% RSLogix 500 project Sesion12_Tarea1_Josue Santana Robledo Corona.RSS, saved by version 8.40.00.08 %
PROJECT "UNTITLED"    % processor: MicroLogix 1200 %

PROGRAM FILES
  LAD 2 "MAIN"  7 rungs
  LAD 3 "ENTRADAS"  6 rungs
  LAD 4 "SALIDAS"  6 rungs
  LAD 5 "AUTOMATICO"  17 rungs
  LAD 6 "MANUAL"  6 rungs
  LAD 7 "HMI"  1 rungs
  LAD 8 "ALARMAS"  1 rungs
  LAD 9 "PARPADEOS"  9 rungs
  LAD 10 "RESETS"  7 rungs
  LAD 11 "LS"  3 rungs

DATA FILES
  O0 OUTPUT  4 elements
  I1 INPUT  4 elements
  S2 STATUS  66 elements
  B3 BINARY  5 elements
  T4 TIMER  7 elements
  C5 COUNTER  3 elements
  R6 CONTROL  1 elements
  N7 INTEGER  1 elements
  F8 FLOAT  1 elements

LADDER 2 "MAIN"
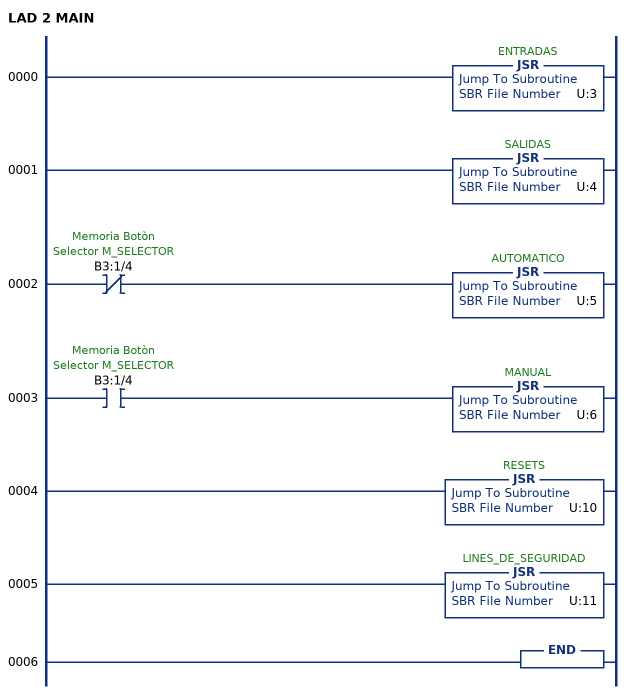
% Rung: 0 %
SOR JSR U:3 EOR
%   U:3  ENTRADAS %
% Rung: 1 %
SOR JSR U:4 EOR
%   U:4  SALIDAS %
% Rung: 2 %
SOR XIO B3:1/4 JSR U:5 EOR
%   B3:1/4  M_SELECTOR  "Memoria Botòn Selector" %
%   U:5  AUTOMATICO %
% Rung: 3 %
SOR XIC B3:1/4 JSR U:6 EOR
%   B3:1/4  M_SELECTOR  "Memoria Botòn Selector" %
%   U:6  MANUAL %
% Rung: 4 %
SOR JSR U:10 EOR
%   U:10  RESETS %
% Rung: 5 %
SOR JSR U:11 EOR
%   U:11  LINES_DE_SEGURIDAD %
% Rung: 6 %
SOR END EOR

LADDER 3 "ENTRADAS"
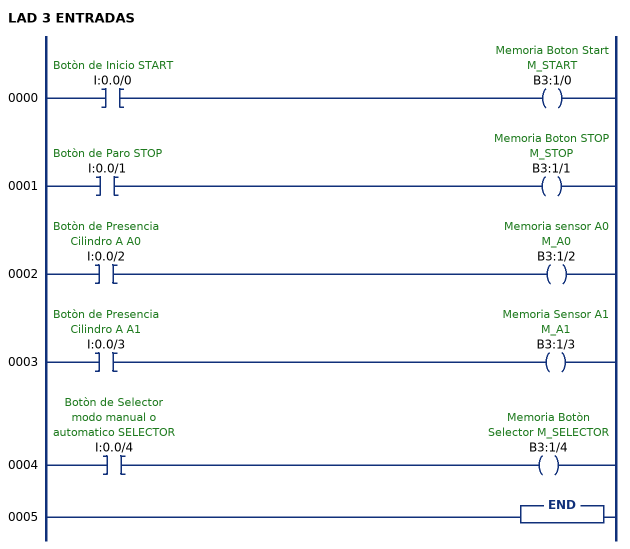
% Rung: 0 %
SOR XIC I:0.0/0 OTE B3:1/0 EOR
%   I:0.0/0  START  "Botòn de Inicio" %
%   B3:1/0  M_START  "Memoria Boton Start" %
% Rung: 1 %
SOR XIC I:0.0/1 OTE B3:1/1 EOR
%   I:0.0/1  STOP  "Botòn de Paro" %
%   B3:1/1  M_STOP  "Memoria Boton STOP" %
% Rung: 2 %
SOR XIC I:0.0/2 OTE B3:1/2 EOR
%   I:0.0/2  A0  "Botòn de Presencia Cilindro A" %
%   B3:1/2  M_A0  "Memoria sensor A0" %
% Rung: 3 %
SOR XIC I:0.0/3 OTE B3:1/3 EOR
%   I:0.0/3  A1  "Botòn de Presencia Cilindro A" %
%   B3:1/3  M_A1  "Memoria Sensor A1" %
% Rung: 4 %
SOR XIC I:0.0/4 OTE B3:1/4 EOR
%   I:0.0/4  SELECTOR  "Botòn de Selector modo manual o automatico" %
%   B3:1/4  M_SELECTOR  "Memoria Botòn Selector" %
% Rung: 5 %
SOR END EOR

LADDER 4 "SALIDAS"
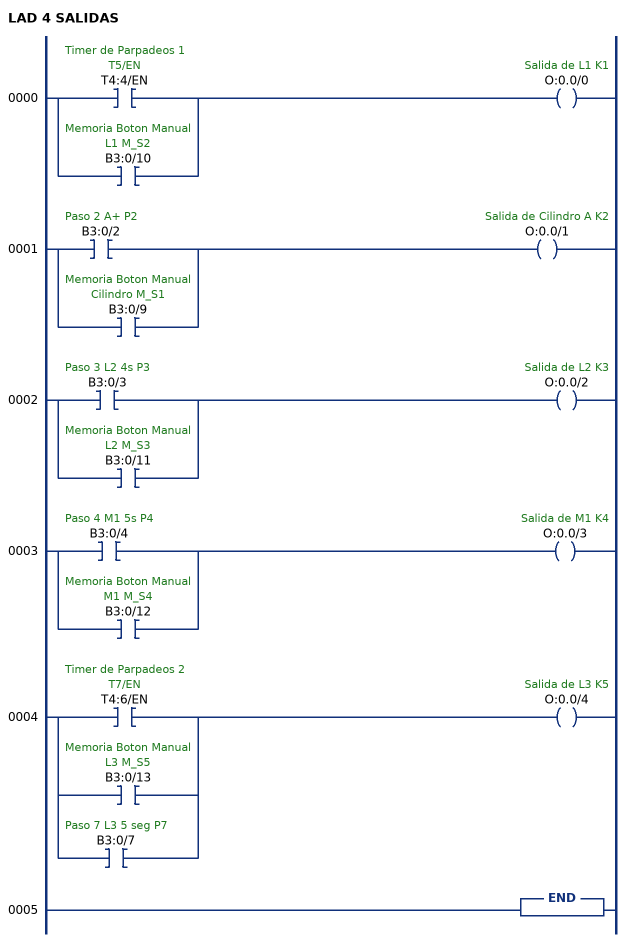
% Rung: 0 %
SOR BST XIC T4:4/EN NXB XIC B3:0/10 BND OTE O:0.0/0 EOR
%   T4:4  T5  "Timer de Parpadeos 1" %
%   B3:0/10  M_S2  "Memoria Boton Manual L1" %
%   O:0.0/0  K1  "Salida de L1" %
% Rung: 1 %
SOR BST XIC B3:0/2 NXB XIC B3:0/9 BND OTE O:0.0/1 EOR
%   B3:0/2  P2  "Paso 2 A+" %
%   B3:0/9  M_S1  "Memoria Boton Manual Cilindro" %
%   O:0.0/1  K2  "Salida de Cilindro A" %
% Rung: 2 %
SOR BST XIC B3:0/3 NXB XIC B3:0/11 BND OTE O:0.0/2 EOR
%   B3:0/3  P3  "Paso 3 L2 4s" %
%   B3:0/11  M_S3  "Memoria Boton Manual L2" %
%   O:0.0/2  K3  "Salida de L2" %
% Rung: 3 %
SOR BST XIC B3:0/4 NXB XIC B3:0/12 BND OTE O:0.0/3 EOR
%   B3:0/4  P4  "Paso 4 M1 5s" %
%   B3:0/12  M_S4  "Memoria Boton Manual M1" %
%   O:0.0/3  K4  "Salida de M1" %
% Rung: 4 %
SOR BST XIC T4:6/EN NXB XIC B3:0/13 NXB XIC B3:0/7 BND OTE O:0.0/4 EOR
%   T4:6  T7  "Timer de Parpadeos 2" %
%   B3:0/13  M_S5  "Memoria Boton Manual L3" %
%   B3:0/7  P7  "Paso 7 L3 5 seg" %
%   O:0.0/4  K5  "Salida de L3" %
% Rung: 5 %
SOR END EOR

LADDER 5 "AUTOMATICO"
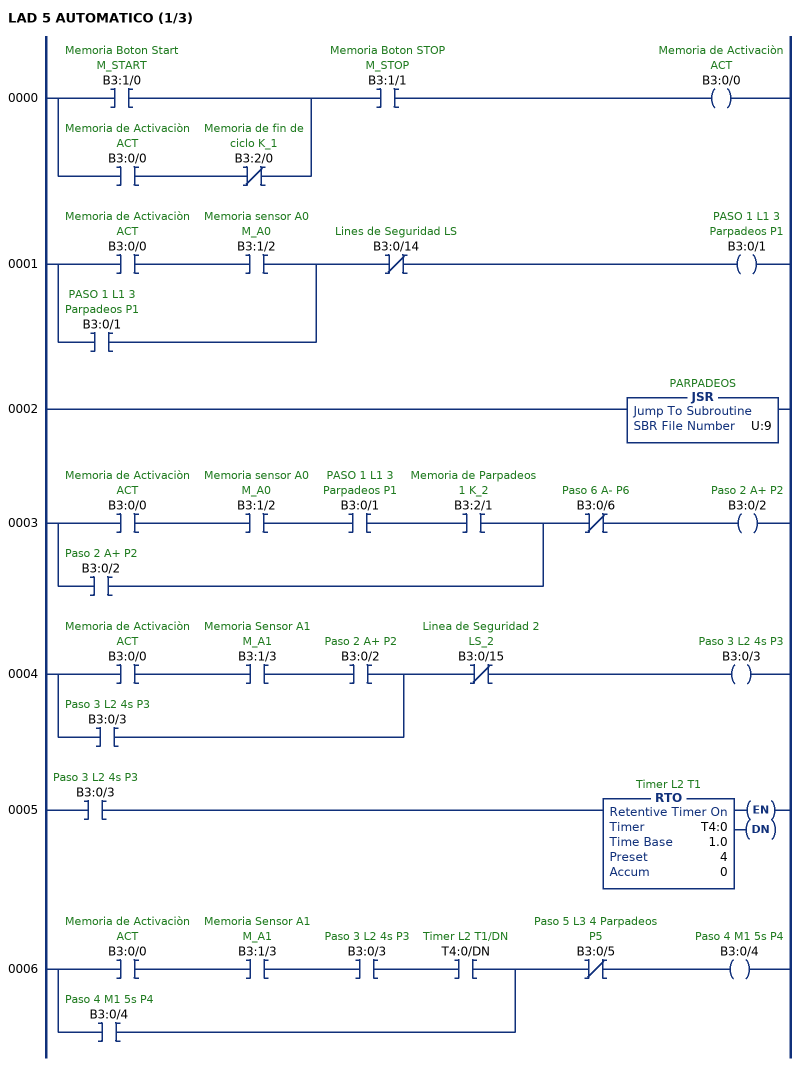
% Rung: 0 %
SOR BST XIC B3:1/0 NXB XIC B3:0/0 XIO B3:2/0 BND XIC B3:1/1 OTE B3:0/0 EOR
%   B3:1/0  M_START  "Memoria Boton Start" %
%   B3:0/0  ACT  "Memoria de Activaciòn" %
%   B3:2/0  K_1  "Memoria de fin de ciclo" %
%   B3:1/1  M_STOP  "Memoria Boton STOP" %
% Rung: 1 %
SOR BST XIC B3:0/0 XIC B3:1/2 NXB XIC B3:0/1 BND XIO B3:0/14 OTE B3:0/1 EOR
%   B3:0/0  ACT  "Memoria de Activaciòn" %
%   B3:1/2  M_A0  "Memoria sensor A0" %
%   B3:0/1  P1  "PASO 1 L1 3 Parpadeos" %
%   B3:0/14  LS  "Lines de Seguridad" %
% Rung: 2 %
SOR JSR U:9 EOR
%   U:9  PARPADEOS %
% Rung: 3 %
SOR BST XIC B3:0/0 XIC B3:1/2 XIC B3:0/1 XIC B3:2/1 NXB XIC B3:0/2 BND XIO B3:0/6 OTE B3:0/2 EOR
%   B3:0/0  ACT  "Memoria de Activaciòn" %
%   B3:1/2  M_A0  "Memoria sensor A0" %
%   B3:0/1  P1  "PASO 1 L1 3 Parpadeos" %
%   B3:2/1  K_2  "Memoria de Parpadeos 1" %
%   B3:0/2  P2  "Paso 2 A+" %
%   B3:0/6  P6  "Paso 6 A-" %
% Rung: 4 %
SOR BST XIC B3:0/0 XIC B3:1/3 XIC B3:0/2 NXB XIC B3:0/3 BND XIO B3:0/15 OTE B3:0/3 EOR
%   B3:0/0  ACT  "Memoria de Activaciòn" %
%   B3:1/3  M_A1  "Memoria Sensor A1" %
%   B3:0/2  P2  "Paso 2 A+" %
%   B3:0/3  P3  "Paso 3 L2 4s" %
%   B3:0/15  LS_2  "Linea de Seguridad 2" %
% Rung: 5 %
SOR XIC B3:0/3 RTO T4:0 1.0 4 0 EOR
%   B3:0/3  P3  "Paso 3 L2 4s" %
%   T4:0  T1  "Timer L2" %
% Rung: 6 %
SOR BST XIC B3:0/0 XIC B3:1/3 XIC B3:0/3 XIC T4:0/DN NXB XIC B3:0/4 BND XIO B3:0/5 OTE B3:0/4 EOR
%   B3:0/0  ACT  "Memoria de Activaciòn" %
%   B3:1/3  M_A1  "Memoria Sensor A1" %
%   B3:0/3  P3  "Paso 3 L2 4s" %
%   T4:0  T1  "Timer L2" %
%   B3:0/4  P4  "Paso 4 M1 5s" %
%   B3:0/5  P5  "Paso 5 L3 4 Parpadeos" %

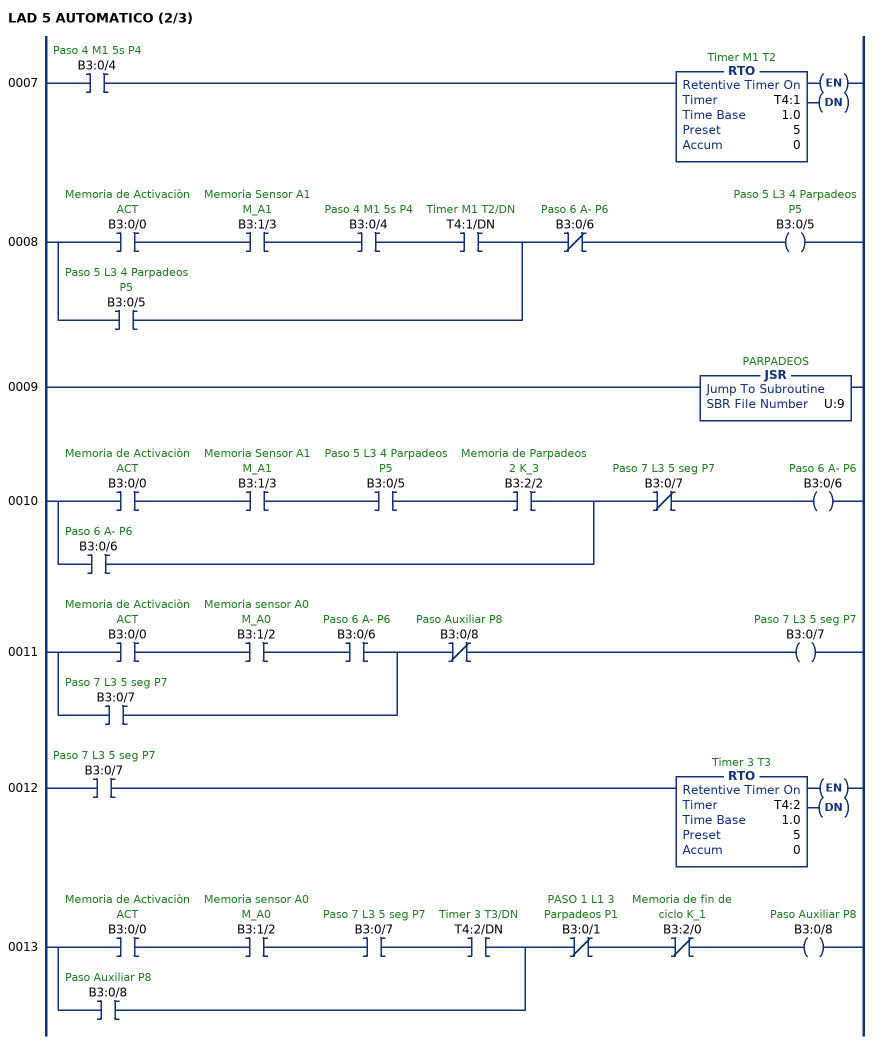
% Rung: 7 %
SOR XIC B3:0/4 RTO T4:1 1.0 5 0 EOR
%   B3:0/4  P4  "Paso 4 M1 5s" %
%   T4:1  T2  "Timer M1" %
% Rung: 8 %
SOR BST XIC B3:0/0 XIC B3:1/3 XIC B3:0/4 XIC T4:1/DN NXB XIC B3:0/5 BND XIO B3:0/6 OTE B3:0/5 EOR
%   B3:0/0  ACT  "Memoria de Activaciòn" %
%   B3:1/3  M_A1  "Memoria Sensor A1" %
%   B3:0/4  P4  "Paso 4 M1 5s" %
%   T4:1  T2  "Timer M1" %
%   B3:0/5  P5  "Paso 5 L3 4 Parpadeos" %
%   B3:0/6  P6  "Paso 6 A-" %
% Rung: 9 %
SOR JSR U:9 EOR
%   U:9  PARPADEOS %
% Rung: 10 %
SOR BST XIC B3:0/0 XIC B3:1/3 XIC B3:0/5 XIC B3:2/2 NXB XIC B3:0/6 BND XIO B3:0/7 OTE B3:0/6 EOR
%   B3:0/0  ACT  "Memoria de Activaciòn" %
%   B3:1/3  M_A1  "Memoria Sensor A1" %
%   B3:0/5  P5  "Paso 5 L3 4 Parpadeos" %
%   B3:2/2  K_3  "Memoria de Parpadeos 2" %
%   B3:0/6  P6  "Paso 6 A-" %
%   B3:0/7  P7  "Paso 7 L3 5 seg" %
% Rung: 11 %
SOR BST XIC B3:0/0 XIC B3:1/2 XIC B3:0/6 NXB XIC B3:0/7 BND XIO B3:0/8 OTE B3:0/7 EOR
%   B3:0/0  ACT  "Memoria de Activaciòn" %
%   B3:1/2  M_A0  "Memoria sensor A0" %
%   B3:0/6  P6  "Paso 6 A-" %
%   B3:0/7  P7  "Paso 7 L3 5 seg" %
%   B3:0/8  P8  "Paso Auxiliar" %
% Rung: 12 %
SOR XIC B3:0/7 RTO T4:2 1.0 5 0 EOR
%   B3:0/7  P7  "Paso 7 L3 5 seg" %
%   T4:2  T3  "Timer 3" %
% Rung: 13 %
SOR BST XIC B3:0/0 XIC B3:1/2 XIC B3:0/7 XIC T4:2/DN NXB XIC B3:0/8 BND XIO B3:0/1 XIO B3:2/0 OTE B3:0/8 EOR
%   B3:0/0  ACT  "Memoria de Activaciòn" %
%   B3:1/2  M_A0  "Memoria sensor A0" %
%   B3:0/7  P7  "Paso 7 L3 5 seg" %
%   T4:2  T3  "Timer 3" %
%   B3:0/8  P8  "Paso Auxiliar" %
%   B3:0/1  P1  "PASO 1 L1 3 Parpadeos" %
%   B3:2/0  K_1  "Memoria de fin de ciclo" %

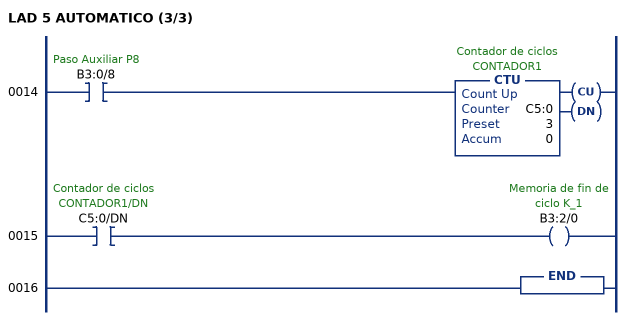
% Rung: 14 %
SOR XIC B3:0/8 CTU C5:0 3 0 EOR
%   B3:0/8  P8  "Paso Auxiliar" %
%   C5:0  CONTADOR1  "Contador de ciclos" %
% Rung: 15 %
SOR XIC C5:0/DN OTE B3:2/0 EOR
%   C5:0  CONTADOR1  "Contador de ciclos" %
%   B3:2/0  K_1  "Memoria de fin de ciclo" %
% Rung: 16 %
SOR END EOR

LADDER 6 "MANUAL"
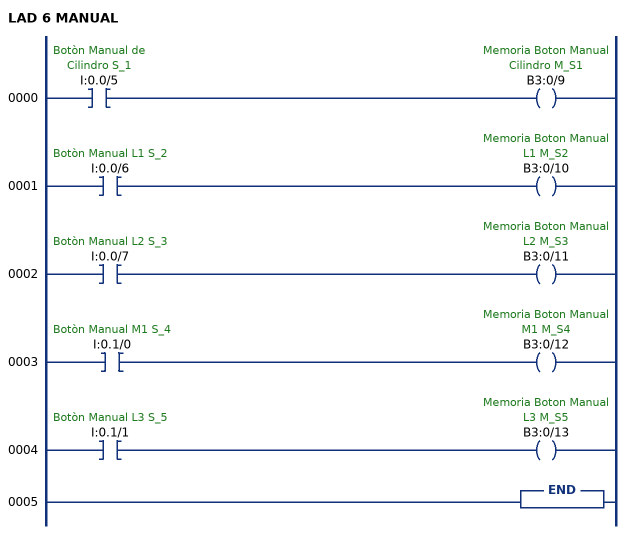
% Rung: 0 %
SOR XIC I:0.0/5 OTE B3:0/9 EOR
%   I:0.0/5  S_1  "Botòn Manual de Cilindro" %
%   B3:0/9  M_S1  "Memoria Boton Manual Cilindro" %
% Rung: 1 %
SOR XIC I:0.0/6 OTE B3:0/10 EOR
%   I:0.0/6  S_2  "Botòn Manual L1" %
%   B3:0/10  M_S2  "Memoria Boton Manual L1" %
% Rung: 2 %
SOR XIC I:0.0/7 OTE B3:0/11 EOR
%   I:0.0/7  S_3  "Botòn Manual L2" %
%   B3:0/11  M_S3  "Memoria Boton Manual L2" %
% Rung: 3 %
SOR XIC I:0.1/0 OTE B3:0/12 EOR
%   I:0.1/0  S_4  "Botòn Manual M1" %
%   B3:0/12  M_S4  "Memoria Boton Manual M1" %
% Rung: 4 %
SOR XIC I:0.1/1 OTE B3:0/13 EOR
%   I:0.1/1  S_5  "Botòn Manual L3" %
%   B3:0/13  M_S5  "Memoria Boton Manual L3" %
% Rung: 5 %
SOR END EOR

LADDER 9 "PARPADEOS"
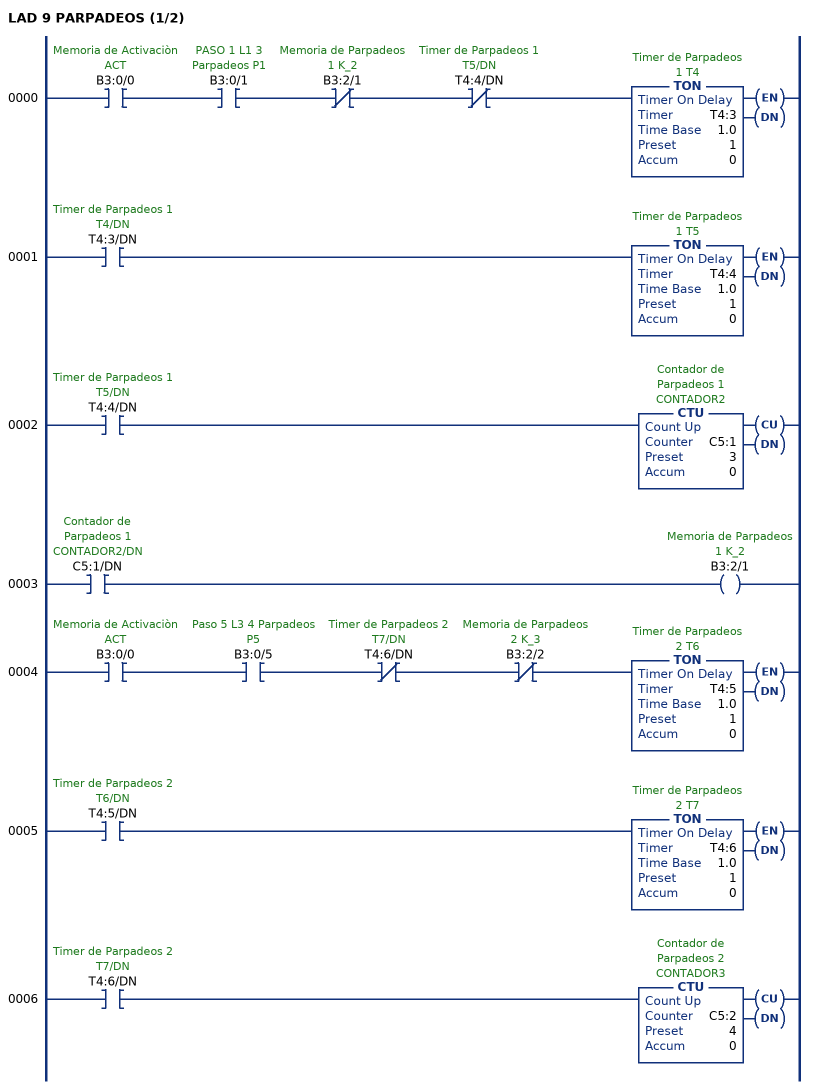
% Rung: 0 %
SOR XIC B3:0/0 XIC B3:0/1 XIO B3:2/1 XIO T4:4/DN TON T4:3 1.0 1 0 EOR
%   B3:0/0  ACT  "Memoria de Activaciòn" %
%   B3:0/1  P1  "PASO 1 L1 3 Parpadeos" %
%   B3:2/1  K_2  "Memoria de Parpadeos 1" %
%   T4:4  T5  "Timer de Parpadeos 1" %
%   T4:3  T4  "Timer de Parpadeos 1" %
% Rung: 1 %
SOR XIC T4:3/DN TON T4:4 1.0 1 0 EOR
%   T4:3  T4  "Timer de Parpadeos 1" %
%   T4:4  T5  "Timer de Parpadeos 1" %
% Rung: 2 %
SOR XIC T4:4/DN CTU C5:1 3 0 EOR
%   T4:4  T5  "Timer de Parpadeos 1" %
%   C5:1  CONTADOR2  "Contador de Parpadeos 1" %
% Rung: 3 %
SOR XIC C5:1/DN OTE B3:2/1 EOR
%   C5:1  CONTADOR2  "Contador de Parpadeos 1" %
%   B3:2/1  K_2  "Memoria de Parpadeos 1" %
% Rung: 4 %
SOR XIC B3:0/0 XIC B3:0/5 XIO T4:6/DN XIO B3:2/2 TON T4:5 1.0 1 0 EOR
%   B3:0/0  ACT  "Memoria de Activaciòn" %
%   B3:0/5  P5  "Paso 5 L3 4 Parpadeos" %
%   T4:6  T7  "Timer de Parpadeos 2" %
%   B3:2/2  K_3  "Memoria de Parpadeos 2" %
%   T4:5  T6  "Timer de Parpadeos 2" %
% Rung: 5 %
SOR XIC T4:5/DN TON T4:6 1.0 1 0 EOR
%   T4:5  T6  "Timer de Parpadeos 2" %
%   T4:6  T7  "Timer de Parpadeos 2" %
% Rung: 6 %
SOR XIC T4:6/DN CTU C5:2 4 0 EOR
%   T4:6  T7  "Timer de Parpadeos 2" %
%   C5:2  CONTADOR3  "Contador de Parpadeos 2" %

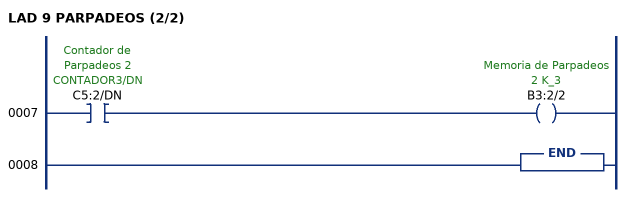
% Rung: 7 %
SOR XIC C5:2/DN OTE B3:2/2 EOR
%   C5:2  CONTADOR3  "Contador de Parpadeos 2" %
%   B3:2/2  K_3  "Memoria de Parpadeos 2" %
% Rung: 8 %
SOR END EOR

LADDER 10 "RESETS"
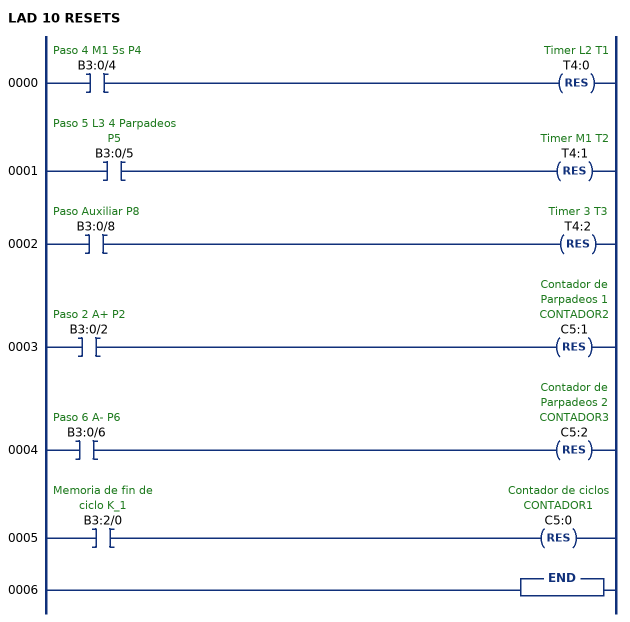
% Rung: 0 %
SOR XIC B3:0/4 RES T4:0 EOR
%   B3:0/4  P4  "Paso 4 M1 5s" %
%   T4:0  T1  "Timer L2" %
% Rung: 1 %
SOR XIC B3:0/5 RES T4:1 EOR
%   B3:0/5  P5  "Paso 5 L3 4 Parpadeos" %
%   T4:1  T2  "Timer M1" %
% Rung: 2 %
SOR XIC B3:0/8 RES T4:2 EOR
%   B3:0/8  P8  "Paso Auxiliar" %
%   T4:2  T3  "Timer 3" %
% Rung: 3 %
SOR XIC B3:0/2 RES C5:1 EOR
%   B3:0/2  P2  "Paso 2 A+" %
%   C5:1  CONTADOR2  "Contador de Parpadeos 1" %
% Rung: 4 %
SOR XIC B3:0/6 RES C5:2 EOR
%   B3:0/6  P6  "Paso 6 A-" %
%   C5:2  CONTADOR3  "Contador de Parpadeos 2" %
% Rung: 5 %
SOR XIC B3:2/0 RES C5:0 EOR
%   B3:2/0  K_1  "Memoria de fin de ciclo" %
%   C5:0  CONTADOR1  "Contador de ciclos" %
% Rung: 6 %
SOR END EOR

LADDER 11 "LS"
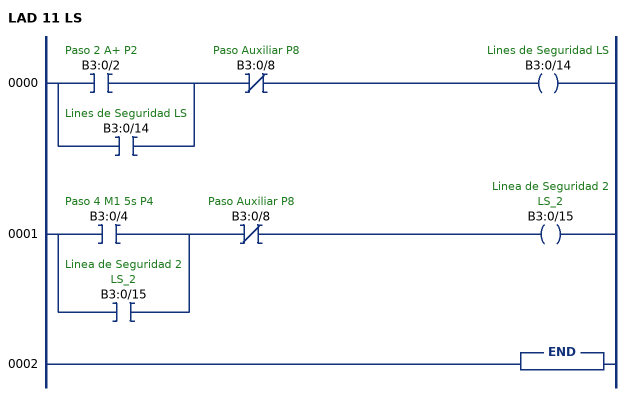
% Rung: 0 %
SOR BST XIC B3:0/2 NXB XIC B3:0/14 BND XIO B3:0/8 OTE B3:0/14 EOR
%   B3:0/2  P2  "Paso 2 A+" %
%   B3:0/14  LS  "Lines de Seguridad" %
%   B3:0/8  P8  "Paso Auxiliar" %
% Rung: 1 %
SOR BST XIC B3:0/4 NXB XIC B3:0/15 BND XIO B3:0/8 OTE B3:0/15 EOR
%   B3:0/4  P4  "Paso 4 M1 5s" %
%   B3:0/15  LS_2  "Linea de Seguridad 2" %
%   B3:0/8  P8  "Paso Auxiliar" %
% Rung: 2 %
SOR END EOR

DATA TABLE (non-zero values as saved)
DATA B3
% B3:0 % 0X0100 0X0006 0X0000 0X0000 0X0000
DATA T4
% .PRE .ACC %
% T4:0 % 4 0
% T4:1 % 5 0
% T4:2 % 5 0
% T4:3 % 1 0
% T4:4 % 1 0
% T4:5 % 1 0
% T4:6 % 1 0
DATA C5
% .PRE .ACC %
% C5:0 % 3 0
% C5:1 % 3 0
% C5:2 % 4 0
